TYPE EtcSlaveBase_82538BE2 :
STRUCT
END_STRUCT
END_TYPE

(* stored: Version 1.2.0.0, ProductVersion 3.1.4024.9
   DUT EtcSlaveBase_82538BE2: Id {07d1b9ec-f5ac-4e81-a079-47416a3af214} *)
